TYPE ST_System_BWK_Parameter :
STRUCT
	AutoQuittierung			: BOOL ;
END_STRUCT
END_TYPE

(* stored: Version 1.1.0.1, ProductVersion 3.1.4024.9
   DUT ST_System_BWK_Parameter: Id {44daed59-6036-40e2-b1a2-e3f48f95d313} *)
